Fanuc KAREL source: NC0076.KL

PROGRAM NC0076
%NOLOCKGROUP
ROUTINE R
VAR
S1:INTEGER
BEGIN
S1=1
WHILE (S1<2) DO
WHILE (S1<2) DO
WHILE (S1<2) DO
WHILE (S1<2) DO
WHILE (S1<2) DO
WHILE (S1<2) DO
WHILE (S1<2) DO
WHILE (S1<2) DO
S1=(S1+1)
ENDWHILE
ENDWHILE
ENDWHILE
ENDWHILE
ENDWHILE
ENDWHILE
ENDWHILE
ENDWHILE
END R
BEGIN
R
END NC0076
